PROGRAM P_JuicePump
VAR
	eState			: ( DISABLED, ENABLED, PUMPING );
	fbPumpSimulator	: FB_JuicePumpSimulator;
	rtStartButton	: R_TRIG;
END_VAR

fbPumpSimulator( bStart := GVL_IO.bPump );

CASE eState OF
	
	DISABLED:
		rtStartButton(CLK := GVL_IO.bStart);
		IF rtStartButton.Q THEN
			eState := ENABLED;
		END_IF
		
	ENABLED:
		GVL_IO.nLedDisplay := GVL_IO.nJuiceSetter;
		
	PUMPING:
		;
		
END_CASE

END_PROGRAM

(* stored: Version 1.1.0.1
   POU P_JuicePump: Id {5fec9547-7f1d-41e1-8d76-841130a6c419}, SpecialFunc None *)
